// TIA Portal V20 export
DATA_BLOCK "ProcedureParameters_DB"   // DB33
AUTHOR : Siemens AG
FAMILY : ServiceControl
VERSION : 1.0
// stored: InstanceOfName ProcedureParameters, InstanceOfType FB
"ProcedureParameters"
   // VAR
   //    MTPAnalog { S7_SetPoint := 'True'} : Array[0..5] of "UDT_MTP_AnaServParam";
   //    MTPDigital { S7_SetPoint := 'True'} : Array[0..0] of "UDT_MTP_DIntServParam";
   //    MTPBinary { S7_SetPoint := 'True'} : Array[0..0] of "UDT_MTP_BinServParam";
   //    MTPString { S7_SetPoint := 'True'} : Array[0..0] of "UDT_MTP_StringServParam";
   // END_VAR
BEGIN
   MTPAnalog[0..4].Sync := True;
   MTPAnalog[0].VExt := 1000.0;
   MTPAnalog[1].VExt := 60.0;
   MTPAnalog[2].VExt := 10.0;
   MTPAnalog[3].VExt := 1500.0;
   MTPAnalog[4].VExt := 60.0;
   MTPAnalog[0].VOp := 1000.0;
   MTPAnalog[1].VOp := 60.0;
   MTPAnalog[2].VOp := 10.0;
   MTPAnalog[3].VOp := 1500.0;
   MTPAnalog[4].VOp := 60.0;
   MTPAnalog[0].VInt := 1000.0;
   MTPAnalog[1].VInt := 60.0;
   MTPAnalog[2].VInt := 10.0;
   MTPAnalog[3].VInt := 1500.0;
   MTPAnalog[4].VInt := 60.0;
   MTPAnalog[0].VReq := 1000.0;
   MTPAnalog[1].VReq := 60.0;
   MTPAnalog[2].VReq := 10.0;
   MTPAnalog[3].VReq := 1500.0;
   MTPAnalog[4].VReq := 60.0;
   MTPAnalog[0].VOut := 1000.0;
   MTPAnalog[1].VOut := 60.0;
   MTPAnalog[2].VOut := 10.0;
   MTPAnalog[3].VOut := 1500.0;
   MTPAnalog[4].VOut := 60.0;
   MTPAnalog[0..4].VSclMin := 0.0;
   MTPAnalog[0].VSclMax := 3000.0;
   MTPAnalog[1].VSclMax := 100.0;
   MTPAnalog[2].VSclMax := 300.0;
   MTPAnalog[3].VSclMax := 2500.0;
   MTPAnalog[4].VSclMax := 300.0;
   MTPAnalog[0].VUnit := 1038;
   MTPAnalog[1].VUnit := 1001;
   MTPAnalog[2].VUnit := 1054;
   MTPAnalog[3].VUnit := 1083;
   MTPAnalog[4].VUnit := 1054;
   MTPAnalog[0].VMin := 5.0;
   MTPAnalog[1].VMin := 10.0;
   MTPAnalog[2].VMin := 5.0;
   MTPAnalog[3].VMin := 0.0;
   MTPAnalog[4].VMin := 5.0;
   MTPAnalog[0].VMax := 3000.0;
   MTPAnalog[1].VMax := 90.0;
   MTPAnalog[2].VMax := 300.0;
   MTPAnalog[3].VMax := 2500.0;
   MTPAnalog[4].VMax := 300.0;
END_DATA_BLOCK
